TYPE ARDeviceErrorSystemLink_t :
STRUCT
	stEventEntity : TcEventEntry;
	callBackPtr : POINTER to bool;
END_STRUCT
END_TYPE

(* stored: Version 1.1.0.1
   DUT ARDeviceErrorSystemLink_t: Id {fed3eb96-8832-490e-a227-6b8a87c31057} *)
